// TIA Portal V20 export
FUNCTION "03 T5 EXCENTRIC Aux" : Void   // FC1318, LAD
TITLE = AUXILIARIES
{ S7_Optimized_Access := 'TRUE' }
// stored: AutoNumber false, SetENOAutomatically false
   VAR_TEMP
      Aux_OS : Bool;
      Aux_sup : Real;
      Aux_inf : Real;
      Aux_DInt : DInt;
      Aux_Real : Real;
   END_VAR
   VAR CONSTANT
      "Max differenza L tubi" : Real := 500.0;
   END_VAR
   VAR_TEMP   // added for the SCL form of the ladder/FBD networks
      _w1 : Bool;
      _w2 : Bool;
   END_VAR
BEGIN

REGION Network 1: =========== MEMORIES ===========
END_REGION

REGION Network 2: Piece presence
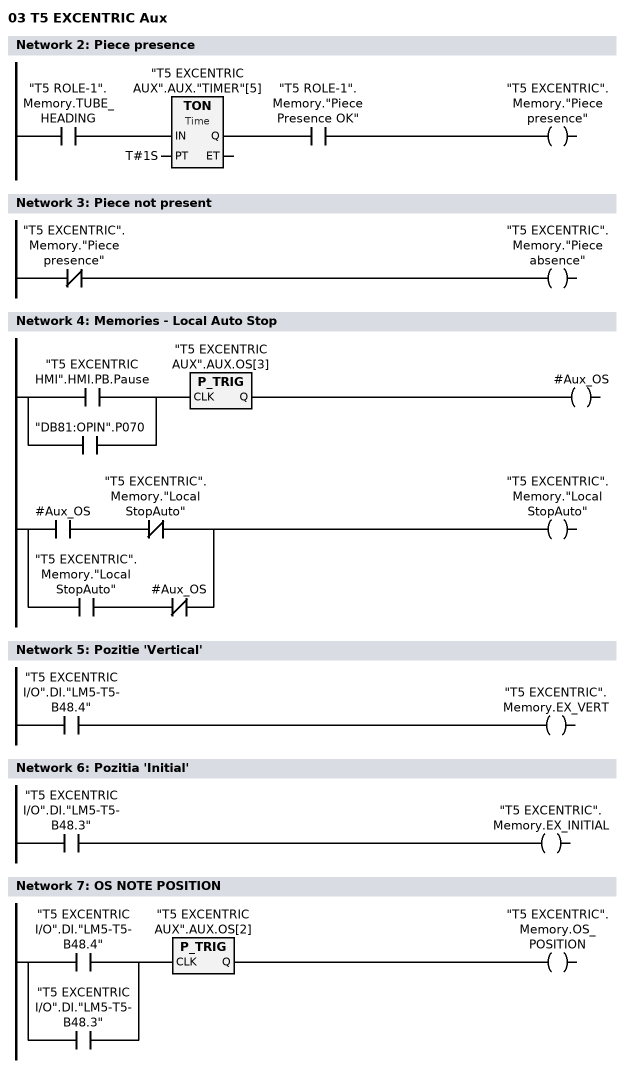
   RUNG wire#powerrail
      Contact( "T5 ROLE-1".Memory.TUBE_HEADING )
      { S7_Templates := "time_type := Time" } "T5 EXCENTRIC AUX".AUX."TIMER"[5].TON(pt := T#1S, et =>)
      Contact( "T5 ROLE-1".Memory."Piece Presence OK" )
      Coil( "T5 EXCENTRIC".Memory."Piece presence" )
   END_RUNG
   // the same network as SCL:
   "T5 EXCENTRIC AUX".AUX."TIMER"[5].TON(IN := "T5 ROLE-1".Memory.TUBE_HEADING, PT := T#1S);
   "T5 EXCENTRIC".Memory."Piece presence" := "T5 EXCENTRIC AUX".AUX."TIMER"[5].Q AND "T5 ROLE-1".Memory."Piece Presence OK";
END_REGION

REGION Network 3: Piece not present
   RUNG wire#powerrail
      I_Contact( "T5 EXCENTRIC".Memory."Piece presence" )
      Coil( "T5 EXCENTRIC".Memory."Piece absence" )
   END_RUNG
   // the same network as SCL:
   "T5 EXCENTRIC".Memory."Piece absence" := NOT "T5 EXCENTRIC".Memory."Piece presence";
END_REGION

REGION Network 4: Memories - Local Auto Stop
   RUNG wire#powerrail
      Contact( "T5 EXCENTRIC HMI".HMI.PB.Pause )
      wire#w1
      P_Trig( "T5 EXCENTRIC AUX".AUX.OS[3] )
      Coil( #Aux_OS )
   END_RUNG
   RUNG wire#powerrail
      Contact( "DB81:OPIN".P070 )
   END_RUNG wire#w1
   RUNG wire#powerrail
      Contact( #Aux_OS )
      I_Contact( "T5 EXCENTRIC".Memory."Local StopAuto" )
      wire#w2
      Coil( "T5 EXCENTRIC".Memory."Local StopAuto" )
   END_RUNG
   RUNG wire#powerrail
      Contact( "T5 EXCENTRIC".Memory."Local StopAuto" )
      I_Contact( #Aux_OS )
   END_RUNG wire#w2
   // the same network as SCL:
   #_w1 := "T5 EXCENTRIC HMI".HMI.PB.Pause OR "DB81:OPIN".P070;
   #_w2 := #_w1 AND NOT "T5 EXCENTRIC AUX".AUX.OS[3];   // rising edge
   "T5 EXCENTRIC AUX".AUX.OS[3] := #_w1;
   #Aux_OS := #_w2;
   "T5 EXCENTRIC".Memory."Local StopAuto" := (#Aux_OS AND NOT "T5 EXCENTRIC".Memory."Local StopAuto") OR ("T5 EXCENTRIC".Memory."Local StopAuto" AND NOT #Aux_OS);
END_REGION

REGION Network 5: Pozitie 'Vertical'
   RUNG wire#powerrail
      Contact( "T5 EXCENTRIC I/O".DI."LM5-T5-B48.4" )
      Coil( "T5 EXCENTRIC".Memory.EX_VERT )
   END_RUNG
   // the same network as SCL:
   "T5 EXCENTRIC".Memory.EX_VERT := "T5 EXCENTRIC I/O".DI."LM5-T5-B48.4";
END_REGION

REGION Network 6: Pozitia 'Initial'
   RUNG wire#powerrail
      Contact( "T5 EXCENTRIC I/O".DI."LM5-T5-B48.3" )
      Coil( "T5 EXCENTRIC".Memory.EX_INITIAL )
   END_RUNG
   // the same network as SCL:
   "T5 EXCENTRIC".Memory.EX_INITIAL := "T5 EXCENTRIC I/O".DI."LM5-T5-B48.3";
END_REGION

REGION Network 7: OS NOTE POSITION
   RUNG wire#powerrail
      Contact( "T5 EXCENTRIC I/O".DI."LM5-T5-B48.4" )
      wire#w1
      P_Trig( "T5 EXCENTRIC AUX".AUX.OS[2] )
      Coil( "T5 EXCENTRIC".Memory.OS_POSITION )
   END_RUNG
   RUNG wire#powerrail
      Contact( "T5 EXCENTRIC I/O".DI."LM5-T5-B48.3" )
   END_RUNG wire#w1
   // the same network as SCL:
   #_w1 := "T5 EXCENTRIC I/O".DI."LM5-T5-B48.4" OR "T5 EXCENTRIC I/O".DI."LM5-T5-B48.3";
   #_w2 := #_w1 AND NOT "T5 EXCENTRIC AUX".AUX.OS[2];   // rising edge
   "T5 EXCENTRIC AUX".AUX.OS[2] := #_w1;
   "T5 EXCENTRIC".Memory.OS_POSITION := #_w2;
END_REGION
END_FUNCTION
